// TIA Portal V16 export
// export: Created 2024-09-05T17:40:15.3450961Z, ExportSetting WithDefaults, DisplayName Totally Integrated Automation Portal, DisplayVersion V16 Update 6, DisplayName TIA Portal Version Control Interface, DisplayVersion V16 Update 2, DisplayName TIA Portal Openness, DisplayVersion V16 Update 6, DisplayName STEP 7 Professional, DisplayVersion V16 Update 6, DisplayName STEP 7 Safety, DisplayVersion V16, DisplayName WinCC Advanced, DisplayVersion V16 Update 6
TYPE "methodListType"
// stored: IsFailsafeCompliant false
   STRUCT
      MethodCount { ExternalAccessible := 'False'; ExternalVisible := 'False'; ExternalWritable := 'False'} : UInt := 0;
      ObjectNodes { ExternalAccessible := 'False'; ExternalVisible := 'False'; ExternalWritable := 'False'; S7_SetPoint := 'True'} : Array[0..0] of OPC_UA_NodeId;
      MethodNodes { ExternalAccessible := 'False'; ExternalVisible := 'False'; ExternalWritable := 'False'; S7_SetPoint := 'True'} : Array[0..0] of OPC_UA_NodeId;
      MethodHdls { ExternalAccessible := 'False'; ExternalVisible := 'False'; ExternalWritable := 'False'} : Array[0..0] of DWord;
   END_STRUCT;
   // ObjectNodes[0].NamespaceIndex := 0;
   // ObjectNodes[0].Identifier := WSTRING#'"OPCMethodSetMachineTime_DB"';
   // ObjectNodes[0].IdentifierType := 1;
   // MethodNodes[0].NamespaceIndex := 0;
   // MethodNodes[0].Identifier := WSTRING#'"OPCMethodSetMachineTime_DB".Method';
   // MethodNodes[0].IdentifierType := 1;
   // MethodHdls[0] := 16#0;
END_TYPE
